// This function has been automatically generated from the project information.
{attribute 'signature_flag' := '1073741824'}
{attribute 'TcGenerated'}
{attribute 'no-analysis'}
FUNCTION F_GetCompany : WSTRING
VAR_INPUT
	
END_VAR

F_GetCompany := "Lisec";

END_FUNCTION

(* stored: Version 1.1.0.1
   POU F_GetCompany: Id {796087cc-ba61-41f4-bdef-c417778a642b}, SpecialFunc None *)
